{attribute 'qualified_only'}
{attribute 'strict'}
{attribute 'to_string'}
TYPE nBottleTypes :
(	
	none := 0,
	first := 1,
	second := 2,
	third :=3
);
END_TYPE

(* stored: Version 1.1.0.1, ProductVersion 3.1.4024.15
   EnumerationTextList nBottleTypes: Id {10188414-6b32-474e-a346-2a2942e03267} *)
